Staubli VAL3: JointFeedback.pjx

--- JointFeedback.pjx ---
Parameters version=s7.7.2 stackSize=5000 millimeterUnit=true
Program file=start.pgx
Program file=stop.pgx
Data file=JointFeedback.dtx

--- JointFeedback.dtx ---
public num nRobotId
public num nValidFields
public num nTime
public num nPositions[10]
public num nVelocities[10]
public num nAccelerations[10]
